// TwinCAT 3 PLC project ExperimentSequencer
// ProgramVersion: 3.1.4026.24
// libraries:
//   Tc2_Standard, * (Beckhoff Automation GmbH)
//   Tc2_System, * (Beckhoff Automation GmbH)
//   Tc3_Module, * (Beckhoff Automation GmbH)
// project tree:
//   / PlcTask.TcTTO
//   DUTs/ DUT_CommandMailbox.TcDUT, DUT_Heartbeat.TcDUT, DUT_LoggerControl.TcDUT, DUT_LoggerSample.TcDUT, DUT_CommutationOverride.TcDUT, DUT_MotorDriverCommand.TcDUT, DUT_MotorFeedbackSnapshot.TcDUT, DUT_ProtocolParams.TcDUT, DUT_SequencerContext.TcDUT, DUT_SequencerStatus.TcDUT
//   GVLs/ GVL_ExperimentSequencer.TcGVL, GVL_ExperimentLogger.TcGVL
//   POUs/ F_ArchWrap2Pi.TcPOU, FB_DifferentialSweep.TcPOU, FB_ExperimentSequencer.TcPOU, FB_ExperimentLogger.TcPOU, FB_IppCurrentRatio.TcPOU, PRG_ExperimentSequencer.TcPOU, PRG_ExperimentLogger.TcPOU
// real-time tasks:
//   TASK PlcTask1: cycle T#250us, priority 21, ADS port 351
//   TASK PlcTask: cycle T#125us, priority 20, ADS port 350
//   TASK StateTask: cycle T#10ms, priority 1, ADS port 352
// I/O:
//   DEVICE Device 3 (EtherCAT), AmsNetId 192.168.10.3.4.1
//     Term 1 (EK1100) [EK1100 EtherCAT Coupler (2A E-Bus)]
//       Term 2 (EL5042) [EL5042 2Ch. BiSS-C Encoder]
//       Term 9 (EL9011) [EL9011 End Terminal]
//     Drive 7 (XE2) [XE2]
//       modules: Module 1 (Cyclic torque with commutation angle Mode), Module 2 (Cyclic torque with commutation angle Mode)
//     Drive 8 (XE2) [XE2]
//       modules: Module 1 (Cyclic torque with commutation angle Mode), Module 2 (Cyclic torque with commutation angle Mode)
// variable links:
//   ExperimentSequencer/ExperimentSequencer Instance <-> MotorRuntime/MotorRuntime Instance
//     PlcTask Inputs/GVL_ExperimentSequencer.motorFeedback <-> PlcTask Outputs/GVL_MotorRuntimeInternal.Feedback
//     PlcTask Outputs/GVL_ExperimentSequencer.commutationOverride <-> PlcTask Inputs/GVL_MotorRuntimeInternal.CommutationOverride
//     PlcTask Outputs/GVL_ExperimentSequencer.driveCommand <-> PlcTask Inputs/GVL_MotorRuntimeInternal.CommissioningCommand
//   MotorRuntime/MotorRuntime Instance <-> Device 3 (EtherCAT)/Drive 7 (XE2)
//     PlcTask Inputs/PRG_MotorRuntime.copleyActualCurrentCountModule1 <-> Module 1 (Cyclic torque with commutation angle Mode)/Cyclic torque with commutation angle Inputs/Torque actual value
//     PlcTask Inputs/PRG_MotorRuntime.copleyActualCurrentCountModule2 <-> Module 2 (Cyclic torque with commutation angle Mode)/Cyclic torque with commutation angle Inputs/Torque actual value
//     PlcTask Inputs/PRG_MotorRuntime.copleyInputToggle <-> WcState/InputToggle
//     PlcTask Inputs/PRG_MotorRuntime.copleyStatusWordModule1 <-> Module 1 (Cyclic torque with commutation angle Mode)/Cyclic torque with commutation angle Inputs/Status word
//     PlcTask Inputs/PRG_MotorRuntime.copleyStatusWordModule2 <-> Module 2 (Cyclic torque with commutation angle Mode)/Cyclic torque with commutation angle Inputs/Status word
//     PlcTask Inputs/PRG_MotorRuntime.copleyWcState <-> WcState/WcState
//     PlcTask Outputs/PRG_MotorRuntime.copleyCommutationAngleModule1 <-> Module 1 (Cyclic torque with commutation angle Mode)/Cyclic torque with commutation angle Outputs/Commutation angle
//     PlcTask Outputs/PRG_MotorRuntime.copleyCommutationAngleModule2 <-> Module 2 (Cyclic torque with commutation angle Mode)/Cyclic torque with commutation angle Outputs/Commutation angle
//     PlcTask Outputs/PRG_MotorRuntime.copleyControlWordModule1 <-> Module 1 (Cyclic torque with commutation angle Mode)/Cyclic torque with commutation angle Outputs/Control word
//     PlcTask Outputs/PRG_MotorRuntime.copleyControlWordModule2 <-> Module 2 (Cyclic torque with commutation angle Mode)/Cyclic torque with commutation angle Outputs/Control word
//     PlcTask Outputs/PRG_MotorRuntime.copleyTargetTorqueModule1 <-> Module 1 (Cyclic torque with commutation angle Mode)/Cyclic torque with commutation angle Outputs/Target Torque
//     PlcTask Outputs/PRG_MotorRuntime.copleyTargetTorqueModule2 <-> Module 2 (Cyclic torque with commutation angle Mode)/Cyclic torque with commutation angle Outputs/Target Torque
//   MotorRuntime/MotorRuntime Instance <-> Device 3 (EtherCAT)/Drive 8 (XE2)
//     PlcTask Inputs/PRG_MotorRuntime.copleyActualCurrentCountModule3 <-> Module 1 (Cyclic torque with commutation angle Mode)/Cyclic torque with commutation angle Inputs/Torque actual value
//     PlcTask Inputs/PRG_MotorRuntime.copleyActualCurrentCountModule4 <-> Module 2 (Cyclic torque with commutation angle Mode)/Cyclic torque with commutation angle Inputs/Torque actual value
//     PlcTask Inputs/PRG_MotorRuntime.copleyInputToggleDrive2 <-> WcState/InputToggle
//     PlcTask Inputs/PRG_MotorRuntime.copleyStatusWordModule3 <-> Module 1 (Cyclic torque with commutation angle Mode)/Cyclic torque with commutation angle Inputs/Status word
//     PlcTask Inputs/PRG_MotorRuntime.copleyStatusWordModule4 <-> Module 2 (Cyclic torque with commutation angle Mode)/Cyclic torque with commutation angle Inputs/Status word
//     PlcTask Inputs/PRG_MotorRuntime.copleyWcStateDrive2 <-> WcState/WcState
//     PlcTask Outputs/PRG_MotorRuntime.copleyCommutationAngleModule3 <-> Module 1 (Cyclic torque with commutation angle Mode)/Cyclic torque with commutation angle Outputs/Commutation angle
//     PlcTask Outputs/PRG_MotorRuntime.copleyCommutationAngleModule4 <-> Module 2 (Cyclic torque with commutation angle Mode)/Cyclic torque with commutation angle Outputs/Commutation angle
//     PlcTask Outputs/PRG_MotorRuntime.copleyControlWordModule3 <-> Module 1 (Cyclic torque with commutation angle Mode)/Cyclic torque with commutation angle Outputs/Control word
//     PlcTask Outputs/PRG_MotorRuntime.copleyControlWordModule4 <-> Module 2 (Cyclic torque with commutation angle Mode)/Cyclic torque with commutation angle Outputs/Control word
//     PlcTask Outputs/PRG_MotorRuntime.copleyTargetTorqueModule3 <-> Module 1 (Cyclic torque with commutation angle Mode)/Cyclic torque with commutation angle Outputs/Target Torque
//     PlcTask Outputs/PRG_MotorRuntime.copleyTargetTorqueModule4 <-> Module 2 (Cyclic torque with commutation angle Mode)/Cyclic torque with commutation angle Outputs/Target Torque
//   MotorRuntime/MotorRuntime Instance <-> Device 3 (EtherCAT)/Term 1 (EK1100)/Term 2 (EL5042)
//     PlcTask Inputs/PRG_MotorRuntime.encoderError <-> FB Inputs Channel 1/Status/Error
//     PlcTask Inputs/PRG_MotorRuntime.encoderInputToggle <-> WcState/InputToggle
//     PlcTask Inputs/PRG_MotorRuntime.encoderPositionRaw <-> FB Inputs Channel 1/Position
//     PlcTask Inputs/PRG_MotorRuntime.encoderReady <-> FB Inputs Channel 1/Status/Ready
//     PlcTask Inputs/PRG_MotorRuntime.encoderTxPdoState <-> FB Inputs Channel 1/Status/TxPDO State
//     PlcTask Inputs/PRG_MotorRuntime.encoderWcState <-> WcState/WcState
//   MotorRuntime/MotorRuntime Instance <-> TcCOM Objects/Object1 (motor_config)
//     PlcTask Inputs/GVL_MotorRuntime.Command/ControlWord <-> motor_config_Y/controlWord
//     PlcTask Outputs/GVL_MotorRuntime.Status/StatusWord <-> motor_config_U/statusWord
//   MotorRuntime/MotorRuntime Instance <-> TcCOM Objects/Object3 (linear_exp_2025a)
//     PlcTask Inputs/GVL_MotorRuntime.Command/TargetTorque <-> TcModuleOutput/LinearSystem/TargetTorque
//     PlcTask Outputs/GVL_MotorRuntime.Status/PositionActualValue <-> TcModuleInput/LinearSystem/Positionactualvalue
//     PlcTask Outputs/GVL_MotorRuntime.Status/TorqueActualValue <-> TcModuleInput/LinearSystem/Torqueactualvalue1
//     PlcTask Outputs/GVL_MotorRuntime.Status/VelocityActualValue <-> TcModuleInput/LinearSystem/Velocityactualvalue
//   MotorRuntime/MotorRuntime Instance <-> TcCOM Objects/Object3 (linear_exp_tunable_2025a)
//     PlcTask Inputs/GVL_MotorRuntime.Command/TargetTorque <-> TcModuleOutput/linearsystem/TargetTorque
//     PlcTask Outputs/GVL_MotorRuntime.Status/PositionActualValue <-> TcModuleInput/linearsystem/PositionActualValue
//     PlcTask Outputs/GVL_MotorRuntime.Status/TorqueActualValue <-> TcModuleInput/linearsystem/TorqueActualValue
//     PlcTask Outputs/GVL_MotorRuntime.Status/VelocityActualValue <-> TcModuleInput/linearsystem/VelocityActualValue
//   TcCOM Objects/Object1 (motor_config) <-> TcCOM Objects/Object3 (linear_exp_2025a)
//     motor_config_U/servoActivate <-> linear_exp_2025a_Y/servostatus
//   TcCOM Objects/Object1 (motor_config) <-> TcCOM Objects/Object3 (linear_exp_tunable_2025a)
//     motor_config_U/servoActivate <-> linear_exp_tunable_2025a_Y/servostatus

CONFIGURATION ExperimentSequencer
    RESOURCE PLC ON TwinCAT3
        TASK PlcTask(INTERVAL := T#250us, PRIORITY := 21);
        PROGRAM PRG_ExperimentSequencer WITH PlcTask : PRG_ExperimentSequencer;
        PROGRAM PRG_ExperimentLogger WITH PlcTask : PRG_ExperimentLogger;
    END_RESOURCE
END_CONFIGURATION

// ---- DUTs/DUT_CommandMailbox.TcDUT
TYPE DUT_CommandMailbox : STRUCT
    // command_id: 1=prepare_protocol, 2=start_protocol, 3=abort_protocol, 4=reset
    command_id                : UINT;
    request_id                : UDINT;
    lease_id                  : UDINT;
    protocol_id               : UINT;

    last_accepted_request_id  : UDINT;
    last_rejected_request_id  : UDINT;
    rejection_reason          : STRING(80);
END_STRUCT
END_TYPE

// ---- DUTs/DUT_Heartbeat.TcDUT
TYPE DUT_Heartbeat : STRUCT
    lease_id : UDINT;
    counter  : UDINT;
END_STRUCT
END_TYPE

// ---- DUTs/DUT_LoggerControl.TcDUT
TYPE DUT_LoggerControl : STRUCT
    reset          : BOOL;
    capture_enable : BOOL;
END_STRUCT
END_TYPE

// ---- DUTs/DUT_LoggerSample.TcDUT
TYPE DUT_LoggerSample : STRUCT
    sample_index                 : UDINT;
    protocol_id                  : UINT;
    phase_id                     : UINT;
    angle_index                  : UINT;
    protocol2_local_sample_index : UINT;
    t_cycle_s                    : LREAL;
    experiment_angle_rad         : LREAL;
    x_ref_traj_m                 : LREAL;
    encoder_position_raw         : DINT;
    encoder_velocity_raw         : DINT;
    copley_actual_current_count  : INT;
    output_torque_count          : INT;
    fault_id                     : UDINT;
    iq_cmd_count_req_lreal       : LREAL;
    target_current_count_lreal   : LREAL;
END_STRUCT
END_TYPE

// ---- DUTs/DUT_CommutationOverride.TcDUT
TYPE DUT_CommutationOverride : STRUCT
    enable                 : BOOL;
    angle_offset_rad       : LREAL;
    axis_index             : UINT;
END_STRUCT
END_TYPE

// ---- DUTs/DUT_MotorDriverCommand.TcDUT
TYPE DUT_MotorDriverCommand : STRUCT
    ControlWord  : WORD;
    TargetTorque : INT;
END_STRUCT
END_TYPE

// ---- DUTs/DUT_MotorFeedbackSnapshot.TcDUT
TYPE DUT_MotorFeedbackSnapshot : STRUCT
    encoder_position_raw       : DINT;
    encoder_velocity_raw       : DINT;
    copley_statusword          : WORD;
    copley_actual_current_count: INT;
    output_torque_count        : INT;
    fault_id                   : UDINT;
END_STRUCT
END_TYPE

// ---- DUTs/DUT_ProtocolParams.TcDUT
TYPE DUT_ProtocolParams : STRUCT
    axis_index                   : UINT := 1;

    position_raw_zero            : DINT := 0;
    position_zero_m              : LREAL := 0.0;
    position_m_per_count         : LREAL := 1.0e-7;
    velocity_mps_per_count       : LREAL := 1.0e-6;

    x_soft_min_m                 : LREAL := -0.01;
    x_soft_max_m                 : LREAL := 0.01;
    max_velocity_mps             : LREAL := 0.02;

    max_target_count             : INT := 50;
    current_ramp_count_per_s     : LREAL := 500.0;

    task_period_s                : LREAL := 0.00025;
    settle_time_s                : LREAL := 0.05;
    pulse_time_s                 : LREAL := 0.05;
    post_time_s                  : LREAL := 0.05;
    timeout_s                    : LREAL := 10.0;

    angle_start_rad              : LREAL := 0.0;
    angle_step_rad               : LREAL := 0.5235987755982988;
    angle_count                  : UINT := 12;

    protocol2_repeat_count       : UINT := 2;
    protocol2_vmax_mps           : LREAL := 0.002;
    protocol2_accel_time_s       : LREAL := 0.050;
    protocol2_const_time_s       : LREAL := 0.000;
    protocol2_pause_time_s       : LREAL := 0.050;
    speed_kp_count_per_mps       : LREAL := 20000.0;
    speed_ki_count_per_m         : LREAL := 0.0;
    speed_integral_limit_count   : INT := 200;
END_STRUCT
END_TYPE

// ---- DUTs/DUT_SequencerContext.TcDUT
TYPE DUT_SequencerContext : STRUCT
    protocol_id                  : UINT;
    phase_id                     : UINT;
    angle_index                  : UINT;
    protocol2_local_sample_index : UINT;
    experiment_angle_rad         : LREAL;
    x_ref_traj_m                 : LREAL;
    t_cycle_s                    : LREAL;
    fault_id                     : UDINT;
    iq_cmd_count_req_lreal       : LREAL;
    target_current_count_lreal   : LREAL;
END_STRUCT
END_TYPE

// ---- DUTs/DUT_SequencerStatus.TcDUT
TYPE DUT_SequencerStatus : STRUCT
    done               : BOOL;
    fault              : BOOL;
    fault_id           : UDINT;
END_STRUCT
END_TYPE

// ---- GVLs/GVL_ExperimentSequencer.TcGVL
{attribute 'qualified_only'}
VAR_GLOBAL
    // ADS commissioning boundary.
    command        : DUT_CommandMailbox;
    protocolParams : DUT_ProtocolParams;
    heartbeat      : DUT_Heartbeat;
    status         : DUT_SequencerStatus;
    // Actual assigned TwinCAT task period. MATLAB reads this value so its
    // timing and analysis stay aligned when switching between 4 and 8 kHz.
    taskPeriod_s   : LREAL;

    // In-project logger inputs.
    context        : DUT_SequencerContext;
    loggerControl  : DUT_LoggerControl;

    // Private commissioning/maintenance link to MotorRuntime. This is not the
    // public virtual-CST interface and remains heartbeat-gated by the sequencer.
    driveCommand        AT %Q* : DUT_MotorDriverCommand;
    commutationOverride AT %Q* : DUT_CommutationOverride;

    // Selected-axis maintenance feedback used only by commissioning and logging.
    motorFeedback  AT %I* : DUT_MotorFeedbackSnapshot;
END_VAR

// ---- GVLs/GVL_ExperimentLogger.TcGVL
{attribute 'qualified_only'}
VAR_GLOBAL CONSTANT
    LOG_CAPACITY : UDINT := 820000;
END_VAR

VAR_GLOBAL
    // ADS read-only download boundary for MATLAB.
    buffer        : ARRAY[0..819999] OF DUT_LoggerSample;
    sampleCount   : UDINT;
    overflow      : BOOL;
END_VAR

// ---- POUs/PRG_ExperimentSequencer.TcPOU
PROGRAM PRG_ExperimentSequencer
VAR
    fbSequencer  : FB_ExperimentSequencer;
    taskIndex      : DINT;
    cycleTime100ns : UDINT;
    taskPeriod_s   : LREAL := 0.00025;
END_VAR

taskIndex := GETCURTASKINDEXEX();
IF taskIndex > 0 THEN
    cycleTime100ns := TwinCAT_SystemInfoVarList._TaskInfo[taskIndex].CycleTime;
    IF cycleTime100ns > 0 THEN
        taskPeriod_s := UDINT_TO_LREAL(cycleTime100ns) * 1.0E-7;
    END_IF
END_IF
GVL_ExperimentSequencer.taskPeriod_s := taskPeriod_s;

fbSequencer(
    TaskPeriod_s := taskPeriod_s,
    Heartbeat := GVL_ExperimentSequencer.heartbeat,
    MotorFeedback := GVL_ExperimentSequencer.motorFeedback,
    Command := GVL_ExperimentSequencer.command,
    ProtocolParams := GVL_ExperimentSequencer.protocolParams);

GVL_ExperimentSequencer.driveCommand := fbSequencer.DriveCommand;
GVL_ExperimentSequencer.commutationOverride := fbSequencer.CommutationOverride;
GVL_ExperimentSequencer.loggerControl := fbSequencer.LoggerControl;
GVL_ExperimentSequencer.context := fbSequencer.Context;
GVL_ExperimentSequencer.status := fbSequencer.Status;

END_PROGRAM

// ---- POUs/FB_ExperimentSequencer.TcPOU
FUNCTION_BLOCK FB_ExperimentSequencer
VAR_INPUT
    TaskPeriod_s       : LREAL := 0.00025;
    HeartbeatTimeout_s : LREAL := 0.150;
    Heartbeat          : DUT_Heartbeat;
    MotorFeedback      : DUT_MotorFeedbackSnapshot;
END_VAR
VAR_IN_OUT
    Command            : DUT_CommandMailbox;
    ProtocolParams     : DUT_ProtocolParams;
END_VAR
VAR_OUTPUT
    DriveCommand       : DUT_MotorDriverCommand;
    CommutationOverride : DUT_CommutationOverride;
    LoggerControl      : DUT_LoggerControl;
    Context            : DUT_SequencerContext;
    Status             : DUT_SequencerStatus;
END_VAR
VAR
    fbDiff             : FB_DifferentialSweep;
    fbIpp              : FB_IppCurrentRatio;
    fbQAxis            : FB_DifferentialSweep;

    state              : UINT;
    lastRequestId      : UDINT;
    lastHeartbeatCtr   : UDINT;
    heartbeatAge_s     : LREAL;
    activeLeaseId      : UDINT;
    activeProtocolId   : UINT;
    activeParams       : DUT_ProtocolParams;
    runTime_s          : LREAL;
    targetRampCount    : INT;
    targetRampLreal    : LREAL;
    rampDelta          : LREAL;
    appliedCommandLreal : LREAL;
    protocolDone       : BOOL;
    protocolFault      : BOOL;
    protocolFaultId    : UDINT;
    protocolBusy       : BOOL;
    iqReq              : INT;
    iqReqLreal         : LREAL;
    phaseId            : UINT;
    angleIndex         : UINT;
    localSampleIndex   : UINT;
    expAngle           : LREAL;
    xRefTraj           : LREAL;
    xAbs_m             : LREAL;
    vActual_mps        : LREAL;
    faultId            : UDINT;
    latchedFaultId     : UDINT;
END_VAR

LoggerControl.reset := FALSE;
LoggerControl.capture_enable := FALSE;
faultId := 0;

IF Heartbeat.lease_id = activeLeaseId THEN
    IF Heartbeat.counter <> lastHeartbeatCtr THEN
        heartbeatAge_s := 0.0;
        lastHeartbeatCtr := Heartbeat.counter;
    ELSE
        heartbeatAge_s := heartbeatAge_s + TaskPeriod_s;
    END_IF
ELSIF state = 2 THEN
    heartbeatAge_s := heartbeatAge_s + TaskPeriod_s;
END_IF

IF Command.request_id <> lastRequestId THEN
    lastRequestId := Command.request_id;
    Command.rejection_reason := '';

    IF Command.command_id = 4 THEN
        state := 0;
        activeLeaseId := 0;
        activeProtocolId := 0;
        targetRampCount := 0;
        targetRampLreal := 0.0;
        heartbeatAge_s := 0.0;
        latchedFaultId := 0;
        LoggerControl.reset := TRUE;
        Command.last_accepted_request_id := Command.request_id;

    ELSIF Command.command_id = 1 THEN
        IF state <> 0 THEN
            Command.last_rejected_request_id := Command.request_id;
            Command.rejection_reason := 'not idle';
        ELSIF (Command.protocol_id < 1) OR (Command.protocol_id > 3) THEN
            Command.last_rejected_request_id := Command.request_id;
            Command.rejection_reason := 'unsupported protocol';
        ELSIF Command.lease_id = 0 THEN
            Command.last_rejected_request_id := Command.request_id;
            Command.rejection_reason := 'zero lease';
        ELSE
            activeParams := ProtocolParams;
            activeParams.task_period_s := TaskPeriod_s;
            IF Command.protocol_id = 3 THEN
                activeParams.angle_count := 1;
                activeParams.angle_start_rad := 0.0;
                activeParams.angle_step_rad := 0.0;
            END_IF
            state := 1;
            activeLeaseId := Command.lease_id;
            activeProtocolId := Command.protocol_id;
            targetRampCount := 0;
            targetRampLreal := 0.0;
            runTime_s := 0.0;
            heartbeatAge_s := 0.0;
            latchedFaultId := 0;
            LoggerControl.reset := TRUE;
            Command.last_accepted_request_id := Command.request_id;
        END_IF

    ELSIF Command.command_id = 2 THEN
        IF (state = 1) AND (Command.lease_id = activeLeaseId) THEN
            state := 2;
            runTime_s := 0.0;
            heartbeatAge_s := 0.0;
            Command.last_accepted_request_id := Command.request_id;
        ELSE
            Command.last_rejected_request_id := Command.request_id;
            Command.rejection_reason := 'not prepared or lease mismatch';
        END_IF

    ELSIF Command.command_id = 3 THEN
        state := 0;
        targetRampCount := 0;
        targetRampLreal := 0.0;
        latchedFaultId := 0;
        Command.last_accepted_request_id := Command.request_id;

    ELSE
        Command.last_rejected_request_id := Command.request_id;
        Command.rejection_reason := 'unknown command';
    END_IF
END_IF

xAbs_m :=
    activeParams.position_zero_m
    + DINT_TO_LREAL(MotorFeedback.encoder_position_raw - activeParams.position_raw_zero)
      * activeParams.position_m_per_count;
vActual_mps := DINT_TO_LREAL(MotorFeedback.encoder_velocity_raw)
    * activeParams.velocity_mps_per_count;

protocolDone := FALSE;
protocolFault := FALSE;
protocolFaultId := 0;
protocolBusy := FALSE;
iqReq := 0;
iqReqLreal := 0.0;
phaseId := 0;
angleIndex := 0;
localSampleIndex := 0;
expAngle := 0.0;
xRefTraj := xAbs_m;

fbDiff(
    enable := (state = 2) AND (activeProtocolId = 1),
    stParams := activeParams,
    x_abs_m := xAbs_m,
    negate_second_pulse := FALSE);

fbIpp(
    enable := (state = 2) AND (activeProtocolId = 2),
    stParams := activeParams,
    x_abs_m := xAbs_m,
    v_actual_mps := vActual_mps);

fbQAxis(
    enable := (state = 2) AND (activeProtocolId = 3),
    stParams := activeParams,
    x_abs_m := xAbs_m,
    negate_second_pulse := TRUE);

IF activeProtocolId = 1 THEN
    protocolBusy := fbDiff.busy;
    protocolDone := fbDiff.done;
    protocolFault := fbDiff.fault;
    protocolFaultId := fbDiff.fault_id;
    iqReq := fbDiff.iq_cmd_count_req;
    iqReqLreal := INT_TO_LREAL(iqReq);
    phaseId := fbDiff.phase_id;
    angleIndex := fbDiff.angle_index;
    expAngle := fbDiff.experiment_angle_rad;
    xRefTraj := fbDiff.x_ref_traj_m;
ELSIF activeProtocolId = 2 THEN
    protocolBusy := fbIpp.busy;
    protocolDone := fbIpp.done;
    protocolFault := fbIpp.fault;
    protocolFaultId := fbIpp.fault_id;
    iqReq := fbIpp.iq_cmd_count_req;
    iqReqLreal := fbIpp.iq_cmd_count_req_lreal;
    phaseId := fbIpp.phase_id;
    angleIndex := fbIpp.angle_index;
    localSampleIndex := fbIpp.protocol2_local_sample_index;
    expAngle := fbIpp.experiment_angle_rad;
    xRefTraj := fbIpp.x_ref_traj_m;
ELSIF activeProtocolId = 3 THEN
    protocolBusy := fbQAxis.busy;
    protocolDone := fbQAxis.done;
    protocolFault := fbQAxis.fault;
    protocolFaultId := fbQAxis.fault_id;
    iqReq := fbQAxis.iq_cmd_count_req;
    iqReqLreal := INT_TO_LREAL(iqReq);
    phaseId := fbQAxis.phase_id;
    angleIndex := fbQAxis.angle_index;
    expAngle := fbQAxis.experiment_angle_rad;
    xRefTraj := fbQAxis.x_ref_traj_m;
END_IF

IF state = 2 THEN
    runTime_s := runTime_s + TaskPeriod_s;
    IF heartbeatAge_s > HeartbeatTimeout_s THEN
        state := 9;
        faultId := 700;
    ELSIF MotorFeedback.fault_id <> 0 THEN
        state := 9;
        faultId := MotorFeedback.fault_id;
    ELSIF protocolFault THEN
        state := 9;
        faultId := protocolFaultId;
    ELSIF (activeParams.timeout_s > 0.0) AND (runTime_s > activeParams.timeout_s) THEN
        state := 9;
        faultId := 701;
    ELSIF (xAbs_m < activeParams.x_soft_min_m) OR (xAbs_m > activeParams.x_soft_max_m) THEN
        state := 9;
        faultId := 702;
    ELSIF ABS(vActual_mps) > activeParams.max_velocity_mps THEN
        state := 9;
        faultId := 703;
    ELSIF protocolDone THEN
        state := 3;
    END_IF
END_IF

IF (state = 9) AND (faultId <> 0) THEN
    latchedFaultId := faultId;
END_IF

IF state <> 2 THEN
    iqReq := 0;
    iqReqLreal := 0.0;
END_IF

rampDelta := activeParams.current_ramp_count_per_s * TaskPeriod_s;
IF rampDelta <= 0.0 THEN
    rampDelta := INT_TO_LREAL(activeParams.max_target_count);
END_IF

IF targetRampLreal < iqReqLreal THEN
    targetRampLreal := targetRampLreal + rampDelta;
    IF targetRampLreal > iqReqLreal THEN
        targetRampLreal := iqReqLreal;
    END_IF
ELSIF targetRampLreal > iqReqLreal THEN
    targetRampLreal := targetRampLreal - rampDelta;
    IF targetRampLreal < iqReqLreal THEN
        targetRampLreal := iqReqLreal;
    END_IF
END_IF
targetRampCount := LREAL_TO_INT(targetRampLreal);
appliedCommandLreal := 0.0;

DriveCommand.ControlWord := WORD#16#0000;
DriveCommand.TargetTorque := 0;

CommutationOverride.enable := FALSE;
CommutationOverride.angle_offset_rad := expAngle;
CommutationOverride.axis_index := activeParams.axis_index;

IF (state = 2) AND protocolBusy AND (heartbeatAge_s <= HeartbeatTimeout_s) THEN
    appliedCommandLreal := targetRampLreal;

    IF (MotorFeedback.copley_statusword AND WORD#16#006F) = WORD#16#0027 THEN
        DriveCommand.ControlWord := WORD#16#000F;
    ELSIF (MotorFeedback.copley_statusword AND WORD#16#006F) = WORD#16#0023 THEN
        DriveCommand.ControlWord := WORD#16#000F;
    ELSIF (MotorFeedback.copley_statusword AND WORD#16#006F) = WORD#16#0021 THEN
        DriveCommand.ControlWord := WORD#16#0007;
    ELSIF (MotorFeedback.copley_statusword AND WORD#16#004F) = WORD#16#0040 THEN
        DriveCommand.ControlWord := WORD#16#0006;
    ELSE
        DriveCommand.ControlWord := WORD#16#0006;
    END_IF
    DriveCommand.TargetTorque := targetRampCount;

    CommutationOverride.enable := TRUE;
    CommutationOverride.angle_offset_rad := expAngle;
END_IF

LoggerControl.capture_enable := (state = 2);

Context.protocol_id := activeProtocolId;
Context.phase_id := phaseId;
Context.angle_index := angleIndex;
Context.protocol2_local_sample_index := localSampleIndex;
Context.experiment_angle_rad := expAngle;
Context.x_ref_traj_m := xRefTraj;
Context.t_cycle_s := runTime_s;
IF state = 9 THEN
    Context.fault_id := latchedFaultId;
ELSE
    Context.fault_id := faultId;
END_IF
Context.iq_cmd_count_req_lreal := iqReqLreal;
Context.target_current_count_lreal := appliedCommandLreal;

Status.done := state = 3;
Status.fault := state = 9;
IF state = 9 THEN
    IF latchedFaultId = 0 THEN
        Status.fault_id := 799;
    ELSE
        Status.fault_id := latchedFaultId;
    END_IF
ELSIF state = 0 THEN
    Status.fault_id := 0;
END_IF

END_FUNCTION_BLOCK

// ---- POUs/FB_DifferentialSweep.TcPOU
FUNCTION_BLOCK FB_DifferentialSweep
VAR_INPUT
    enable              : BOOL;
    stParams            : DUT_ProtocolParams;
    x_abs_m             : LREAL;
    negate_second_pulse : BOOL := FALSE;
END_VAR
VAR_OUTPUT
    busy                : BOOL;
    done                : BOOL;
    fault               : BOOL;
    fault_id            : UDINT;
    iq_cmd_count_req    : INT;
    experiment_angle_rad: LREAL;
    phase_id            : UINT;
    angle_index         : UINT;
    x_ref_traj_m        : LREAL;
END_VAR
VAR
    wasEnabled          : BOOL;
    tPhase_s            : LREAL;
    alpha               : LREAL;
END_VAR

IF NOT enable THEN
    wasEnabled := FALSE;
    tPhase_s := 0.0;
    busy := FALSE;
    done := FALSE;
    fault := FALSE;
    fault_id := 0;
    iq_cmd_count_req := 0;
    experiment_angle_rad := 0.0;
    phase_id := 0;
    angle_index := 0;
    x_ref_traj_m := x_abs_m;
    RETURN;
END_IF

IF NOT wasEnabled THEN
    wasEnabled := TRUE;
    busy := TRUE;
    done := FALSE;
    fault := FALSE;
    fault_id := 0;
    tPhase_s := 0.0;
    phase_id := 0;
    angle_index := 0;
END_IF

IF (stParams.angle_count = 0)
    OR (negate_second_pulse AND (stParams.max_target_count <= 0)) THEN
    fault := TRUE;
    fault_id := 100;
    busy := FALSE;
    iq_cmd_count_req := 0;
    RETURN;
END_IF

alpha := stParams.angle_start_rad + UINT_TO_LREAL(angle_index) * stParams.angle_step_rad;
x_ref_traj_m := x_abs_m;
iq_cmd_count_req := 0;
experiment_angle_rad := alpha;

CASE phase_id OF
0:
    iq_cmd_count_req := 0;
    IF tPhase_s >= stParams.settle_time_s THEN
        phase_id := 1;
        tPhase_s := 0.0;
    END_IF

1:
    experiment_angle_rad := alpha;
    iq_cmd_count_req := stParams.max_target_count;
    IF tPhase_s >= stParams.pulse_time_s THEN
        phase_id := 2;
        tPhase_s := 0.0;
    END_IF

2:
    iq_cmd_count_req := 0;
    IF tPhase_s >= stParams.settle_time_s THEN
        phase_id := 3;
        tPhase_s := 0.0;
    END_IF

3:
    IF negate_second_pulse THEN
        iq_cmd_count_req := -stParams.max_target_count;
    ELSE
        experiment_angle_rad := F_ArchWrap2Pi(alpha + 3.14159265358979323846);
        iq_cmd_count_req := stParams.max_target_count;
    END_IF
    IF tPhase_s >= stParams.pulse_time_s THEN
        phase_id := 4;
        tPhase_s := 0.0;
    END_IF

4:
    iq_cmd_count_req := 0;
    IF tPhase_s >= stParams.post_time_s THEN
        IF angle_index + 1 >= stParams.angle_count THEN
            busy := FALSE;
            done := TRUE;
        ELSE
            angle_index := angle_index + 1;
            phase_id := 0;
            tPhase_s := 0.0;
        END_IF
    END_IF
ELSE
    fault := TRUE;
    fault_id := 400;
    busy := FALSE;
END_CASE

IF busy THEN
    tPhase_s := tPhase_s + stParams.task_period_s;
END_IF

END_FUNCTION_BLOCK

// ---- POUs/F_ArchWrap2Pi.TcPOU
FUNCTION F_ArchWrap2Pi : LREAL
VAR_INPUT
    theta : LREAL;
END_VAR
VAR CONSTANT
    TWO_PI : LREAL := 6.2831853071795864769;
END_VAR
VAR
    y : LREAL;
END_VAR

y := theta - TWO_PI * LREAL_TO_DINT(theta / TWO_PI);
WHILE y < 0.0 DO
    y := y + TWO_PI;
END_WHILE
WHILE y >= TWO_PI DO
    y := y - TWO_PI;
END_WHILE
F_ArchWrap2Pi := y;

END_FUNCTION

// ---- POUs/FB_IppCurrentRatio.TcPOU
FUNCTION_BLOCK FB_IppCurrentRatio
VAR_INPUT
    enable              : BOOL;
    stParams            : DUT_ProtocolParams;
    x_abs_m             : LREAL;
    v_actual_mps        : LREAL;
END_VAR
VAR_OUTPUT
    busy                : BOOL;
    done                : BOOL;
    fault               : BOOL;
    fault_id            : UDINT;
    iq_cmd_count_req    : INT;
    iq_cmd_count_req_lreal : LREAL;
    protocol2_local_sample_index : UINT;
    experiment_angle_rad: LREAL;
    phase_id            : UINT;
    angle_index         : UINT;
    x_ref_traj_m        : LREAL;
END_VAR
VAR
    wasEnabled          : BOOL;
    step_id             : UINT;
    repeat_index        : UINT;
    tStep_s             : LREAL;
    xRef                : LREAL;
    vRef                : LREAL;
    vRefCommand         : LREAL;
    speedErr            : LREAL;
    speedInt            : LREAL;
    speedIntLimit       : LREAL;
    iqReq               : LREAL;
    vmax                : LREAL;
    accelTime           : LREAL;
    constTime           : LREAL;
    pauseTime           : LREAL;
    accel               : LREAL;
    taskDt_s            : LREAL;
    localSampleIndex    : UINT;
    prevAngleIndex      : UINT;
    angleJustChanged    : BOOL;
END_VAR

IF NOT enable THEN
    wasEnabled := FALSE;
    step_id := 0;
    repeat_index := 0;
    tStep_s := 0.0;
    speedInt := 0.0;
    busy := FALSE;
    done := FALSE;
    fault := FALSE;
    fault_id := 0;
    iq_cmd_count_req := 0;
    iq_cmd_count_req_lreal := 0.0;
    protocol2_local_sample_index := 0;
    experiment_angle_rad := 0.0;
    phase_id := 0;
    angle_index := 0;
    x_ref_traj_m := x_abs_m;
    localSampleIndex := 0;
    prevAngleIndex := 0;
    angleJustChanged := FALSE;
    RETURN;
END_IF

IF NOT wasEnabled THEN
    wasEnabled := TRUE;
    busy := TRUE;
    done := FALSE;
    fault := FALSE;
    fault_id := 0;
    step_id := 0;
    repeat_index := 0;
    tStep_s := 0.0;
    speedInt := 0.0;
    phase_id := 0;
    angle_index := 0;
    localSampleIndex := 0;
    prevAngleIndex := angle_index;
    angleJustChanged := FALSE;
    xRef := x_abs_m;
    x_ref_traj_m := x_abs_m;
END_IF

taskDt_s := stParams.task_period_s;
vmax := stParams.protocol2_vmax_mps;
accelTime := stParams.protocol2_accel_time_s;
constTime := stParams.protocol2_const_time_s;
pauseTime := stParams.protocol2_pause_time_s;

IF (taskDt_s <= 0.0) OR (vmax <= 0.0) OR (accelTime <= 0.0) OR (pauseTime < 0.0) THEN
    fault := TRUE;
    fault_id := 100;
    busy := FALSE;
    iq_cmd_count_req := 0;
    iq_cmd_count_req_lreal := 0.0;
    protocol2_local_sample_index := 0;
    RETURN;
END_IF

IF angle_index = 0 THEN
    experiment_angle_rad := 0.0;
ELSE
    experiment_angle_rad := -3.14159265358979323846 / 2.0;
END_IF

accel := vmax / accelTime;
vRef := 0.0;
CASE step_id OF
0:
    vRef := accel * tStep_s;
    IF vRef > vmax THEN
        vRef := vmax;
    END_IF
    IF tStep_s >= accelTime THEN
        step_id := 1;
        tStep_s := 0.0;
    END_IF
1:
    vRef := vmax;
    IF constTime <= 0.0 THEN
        step_id := 2;
        tStep_s := 0.0;
    ELSIF tStep_s >= constTime THEN
        step_id := 2;
        tStep_s := 0.0;
    END_IF
2:
    vRef := vmax - accel * tStep_s;
    IF vRef < 0.0 THEN
        vRef := 0.0;
    END_IF
    IF tStep_s >= accelTime THEN
        IF pauseTime <= 0.0 THEN
            step_id := 4;
        ELSE
            step_id := 3;
        END_IF
        tStep_s := 0.0;
        speedInt := 0.0;
    END_IF
3:
    vRef := 0.0;
    IF tStep_s >= pauseTime THEN
        step_id := 4;
        tStep_s := 0.0;
    END_IF
4:
    vRef := -accel * tStep_s;
    IF vRef < -vmax THEN
        vRef := -vmax;
    END_IF
    IF tStep_s >= accelTime THEN
        step_id := 5;
        tStep_s := 0.0;
    END_IF
5:
    vRef := -vmax;
    IF constTime <= 0.0 THEN
        step_id := 6;
        tStep_s := 0.0;
    ELSIF tStep_s >= constTime THEN
        step_id := 6;
        tStep_s := 0.0;
    END_IF
6:
    vRef := -vmax + accel * tStep_s;
    IF vRef > 0.0 THEN
        vRef := 0.0;
    END_IF
    IF tStep_s >= accelTime THEN
        tStep_s := 0.0;
        speedInt := 0.0;
        IF pauseTime <= 0.0 THEN
            step_id := 0;
            IF angle_index = 0 THEN
                angle_index := 1;
            ELSE
                angle_index := 0;
                IF repeat_index + 1 >= stParams.protocol2_repeat_count THEN
                    busy := FALSE;
                    done := TRUE;
                    phase_id := 99;
                ELSE
                    repeat_index := repeat_index + 1;
                END_IF
            END_IF
        ELSE
            step_id := 7;
        END_IF
    END_IF
7:
    vRef := 0.0;
    IF tStep_s >= pauseTime THEN
        step_id := 0;
        tStep_s := 0.0;
        speedInt := 0.0;
        IF angle_index = 0 THEN
            angle_index := 1;
        ELSE
            angle_index := 0;
            IF repeat_index + 1 >= stParams.protocol2_repeat_count THEN
                busy := FALSE;
                done := TRUE;
                phase_id := 99;
            ELSE
                repeat_index := repeat_index + 1;
            END_IF
        END_IF
    END_IF
ELSE
    fault := TRUE;
    fault_id := 400;
    busy := FALSE;
END_CASE

angleJustChanged := angle_index <> prevAngleIndex;
IF angleJustChanged THEN
    localSampleIndex := 0;
    prevAngleIndex := angle_index;
END_IF

protocol2_local_sample_index := localSampleIndex;

IF done THEN
    iq_cmd_count_req := 0;
    iq_cmd_count_req_lreal := 0.0;
    x_ref_traj_m := xRef;
    RETURN;
END_IF

IF stParams.velocity_mps_per_count > 0.0 THEN
    vRefCommand := DINT_TO_LREAL(LREAL_TO_DINT(vRef / stParams.velocity_mps_per_count))
                   * stParams.velocity_mps_per_count;
ELSE
    vRefCommand := vRef;
END_IF
xRef := xRef + vRefCommand * taskDt_s;
x_ref_traj_m := xRef;

IF (step_id = 3) OR (step_id = 7) THEN
    phase_id := 90;
    iq_cmd_count_req := 0;
    iq_cmd_count_req_lreal := 0.0;
ELSE
    IF angle_index = 0 THEN
        phase_id := 10;
    ELSE
        phase_id := 11;
    END_IF

    speedErr := vRefCommand - v_actual_mps;
    IF stParams.speed_ki_count_per_m <> 0.0 THEN
        speedInt := speedInt + speedErr * taskDt_s;
        speedIntLimit := INT_TO_LREAL(stParams.speed_integral_limit_count) / ABS(stParams.speed_ki_count_per_m);
        IF speedInt > speedIntLimit THEN
            speedInt := speedIntLimit;
        ELSIF speedInt < -speedIntLimit THEN
            speedInt := -speedIntLimit;
        END_IF
    ELSE
        speedInt := 0.0;
    END_IF

    iqReq := stParams.speed_kp_count_per_mps * speedErr
             + stParams.speed_ki_count_per_m * speedInt;
    IF iqReq > INT_TO_LREAL(stParams.max_target_count) THEN
        iqReq := INT_TO_LREAL(stParams.max_target_count);
    ELSIF iqReq < -INT_TO_LREAL(stParams.max_target_count) THEN
        iqReq := -INT_TO_LREAL(stParams.max_target_count);
    END_IF
    iq_cmd_count_req_lreal := iqReq;
    iq_cmd_count_req := LREAL_TO_INT(iqReq);
END_IF

IF busy THEN
    tStep_s := tStep_s + taskDt_s;
    IF localSampleIndex < 65535 THEN
        localSampleIndex := localSampleIndex + 1;
    END_IF
END_IF

END_FUNCTION_BLOCK

// ---- POUs/PRG_ExperimentLogger.TcPOU
PROGRAM PRG_ExperimentLogger
VAR
    fbLogger : FB_ExperimentLogger;
END_VAR

fbLogger(
    Control := GVL_ExperimentSequencer.loggerControl,
    Context := GVL_ExperimentSequencer.context,
    MotorFeedback := GVL_ExperimentSequencer.motorFeedback,
    Buffer := GVL_ExperimentLogger.buffer);

GVL_ExperimentLogger.sampleCount := fbLogger.SampleCount;
GVL_ExperimentLogger.overflow := fbLogger.Overflow;

END_PROGRAM

// ---- POUs/FB_ExperimentLogger.TcPOU
FUNCTION_BLOCK FB_ExperimentLogger
VAR_INPUT
    Control       : DUT_LoggerControl;
    Context       : DUT_SequencerContext;
    MotorFeedback : DUT_MotorFeedbackSnapshot;
END_VAR
VAR_IN_OUT
    Buffer        : ARRAY[0..819999] OF DUT_LoggerSample;
END_VAR
VAR_OUTPUT
    SampleCount   : UDINT;
    Overflow      : BOOL;
END_VAR
VAR
    sample        : DUT_LoggerSample;
END_VAR

IF Control.reset THEN
    SampleCount := 0;
    Overflow := FALSE;
    RETURN;
END_IF

IF Control.capture_enable AND NOT Overflow THEN
    IF SampleCount < GVL_ExperimentLogger.LOG_CAPACITY THEN
        sample.sample_index := SampleCount;
        sample.protocol_id := Context.protocol_id;
        sample.phase_id := Context.phase_id;
        sample.angle_index := Context.angle_index;
        sample.protocol2_local_sample_index := Context.protocol2_local_sample_index;
        sample.t_cycle_s := Context.t_cycle_s;
        sample.experiment_angle_rad := Context.experiment_angle_rad;
        sample.x_ref_traj_m := Context.x_ref_traj_m;
        sample.iq_cmd_count_req_lreal := Context.iq_cmd_count_req_lreal;
        sample.target_current_count_lreal := Context.target_current_count_lreal;
        sample.encoder_position_raw := MotorFeedback.encoder_position_raw;
        sample.encoder_velocity_raw := MotorFeedback.encoder_velocity_raw;
        sample.copley_actual_current_count := MotorFeedback.copley_actual_current_count;
        sample.output_torque_count := MotorFeedback.output_torque_count;
        IF MotorFeedback.fault_id <> 0 THEN
            sample.fault_id := MotorFeedback.fault_id;
        ELSE
            sample.fault_id := Context.fault_id;
        END_IF
        Buffer[TO_DINT(SampleCount)] := sample;
        SampleCount := SampleCount + 1;
    ELSE
        Overflow := TRUE;
    END_IF
END_IF

END_FUNCTION_BLOCK
